RoboDK station: deburring.rdk

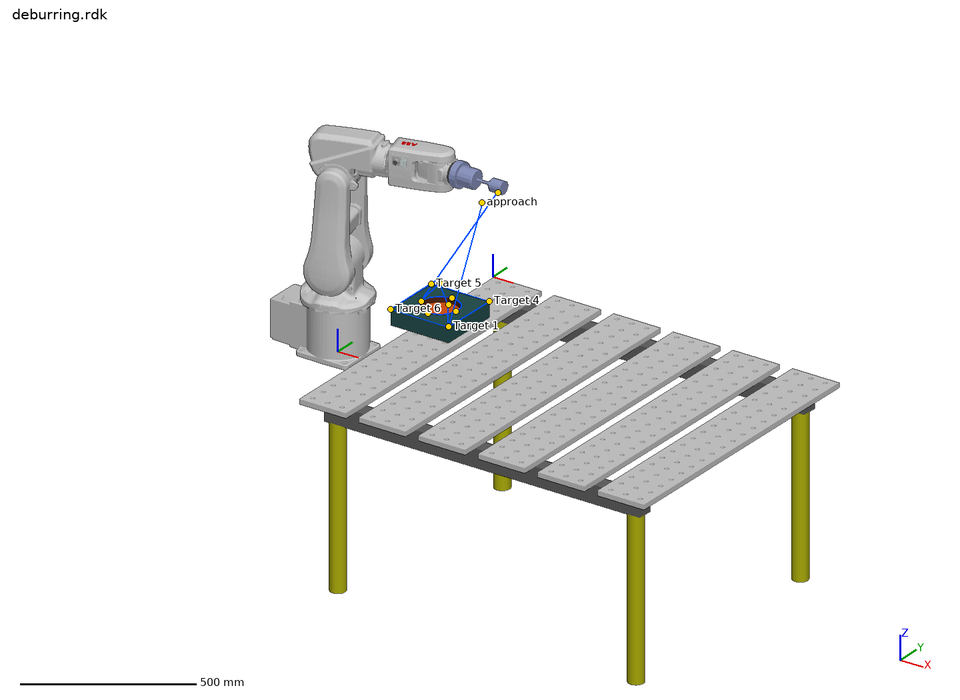
[picture v0: the station drawn from its stored meshes, robots at their saved joint values, targets as dots, program paths as lines]
Station deburring (saved by RoboDK 5.3.4). Poses are relative to the parent item; angles as X-Y-Z fixed-axis rotations.
  - frame ABB IRB 120-3/0.6 Base at (0, 0, 0) mm
    - robot ABB IRB 120-3/0.6: 6 axes, payload 3 kg, reach 580 mm, repeatability 0.01 mm, weight 25 kg
        modified DH rows (alpha deg, a mm, theta deg, d mm): 0, 0, 0, 290; -90, 0, -90, 0; 0, 270, 0, 0; -90, 70, 0, 302; 90, 0, 0, 0; -90, 0, 180, 72
        joint limits [-165, -110, -90, -160, -120, -400] to [165, 110, 70, 160, 120, 400]; home [0, 0, 0, 0, 0, 0]; saved at [14.502, 2.119, -2.154, 90.135, -14.502, -90.14]
      - tool AssemblySpindleSide, TCP at (20, 0, 125) mm, rotated rx 0 ry 45 rz 0 deg, size 80 x 163 x 80 mm
  - object Table at (800, 0, 100) mm, size 1193.8 x 965.2 x 609.6 mm, geometry from welding_table.sld
  - frame worktable at (200, 480, 100) mm
    - object Task2_Part at (60, -590, 100) mm, rotated rx 90 ry 0 rz 0 deg, size 200 x 50 x 200 mm, geometry from Task2_Part.STEP
    - target approach (Cartesian target) at (299, -480, 510) mm, rotated rx -180 ry 45 rz -180 deg; joints [0, 0, 0, 0, 0, 0] of ABB IRB 120-3/0.6
    - target retract (Cartesian target) at (299, -401.89, 510) mm, rotated rx 180 ry 45 rz 180 deg; joints [14.502, 2.119, -2.154, 90.135, -14.502, -90.14] of ABB IRB 120-3/0.6
    - target Target 1 (Cartesian target) at (260, -590, 150) mm, rotated rx 180 ry 0 rz -180 deg; joints [-18.186, 16.881, 24.041, 66.872, 13.885, -79.329] of ABB IRB 120-3/0.6
    - target Target 4 (Cartesian target) at (260, -390, 150) mm, rotated rx -180 ry 0 rz -180 deg; joints [15.045, 15.786, 25.439, -65.976, 11.593, 76.295] of ABB IRB 120-3/0.6
    - target Target 4-5 turning (Cartesian target) at (260, -390, 150) mm, rotated rx 180 ry 0 rz -90 deg; joints [-4.371, 38.309, -6.748, 48.185, 71.084, -116.089] of ABB IRB 120-3/0.6
    - target Target 5 (Cartesian target) at (60, -390, 150) mm, rotated rx -180 ry 0 rz -90 deg; joints [-7.701, -1.111, 44.482, 50.43, 65.373, -127.586] of ABB IRB 120-3/0.6
    - target Target 5-6 turning (Cartesian target) at (60, -390, 150) mm, rotated rx 180 ry 0 rz 0 deg; joints [13.152, 25.112, 12.943, 9.312, 96.103, -169.619] of ABB IRB 120-3/0.6
    - target Target 6 (Cartesian target) at (60, -590, 150) mm, rotated rx 180 ry 0 rz 0 deg; joints [-15.939, 26.08, 11.574, -11.262, 96.105, -192.63] of ABB IRB 120-3/0.6
    - target Target 6-7 turning (Cartesian target) at (60, -590, 150) mm, rotated rx -180 ry 0 rz 90 deg; joints [3.337, -1.525, 44.887, -52.465, 62.898, -234.62] of ABB IRB 120-3/0.6
    - target Target 7 (Cartesian target) at (260, -590, 150) mm, rotated rx -180 ry 0 rz 90 deg; joints [1.887, 38.076, -6.383, -49.021, 69.41, 114.709] of ABB IRB 120-3/0.6
    - target Target 7 protect (Cartesian target) at (260, -590, 220) mm, rotated rx -180 ry 0 rz 90 deg; joints [1.887, 34.449, -14.133, -46.477, 77.076, 105.92] of ABB IRB 120-3/0.6
    - target Target 8 (Cartesian target) at (160, -490, 220) mm, rotated rx -180 ry 0 rz -180 deg; joints [-2.438, -13.888, 41.637, 5.787, 17.359, -7.249] of ABB IRB 120-3/0.6
    - target Target 13 (Cartesian target) at (100.44, -497.23, 150) mm, rotated rx 180 ry 0 rz 180 deg; joints [-5.615, -22.25, 61.415, 33.679, 7.167, -37.448] of ABB IRB 120-3/0.6
    - target Target 17 (Cartesian target) at (219.56, -497.23, 150) mm, rotated rx -180 ry 0 rz 0 deg; joints [-1.812, 60.736, -44.257, -1.458, 118.499, -181.977] of ABB IRB 120-3/0.6
    - target Target 15 (Cartesian target) at (160, -430, 150) mm, rotated rx -180 ry 0 rz 90 deg; joints [25.945, 26.039, 11.631, -40.337, 79.208, 133.566] of ABB IRB 120-3/0.6
    - target Target 16 (Cartesian target) at (160, -550, 150) mm, rotated rx -180 ry 0 rz -90 deg; joints [-28.462, 27.811, 9.093, 38.995, 81.076, -134.635] of ABB IRB 120-3/0.6
  - program prog1 (15 instructions, listed below)
  - program main (1 instructions, listed below)
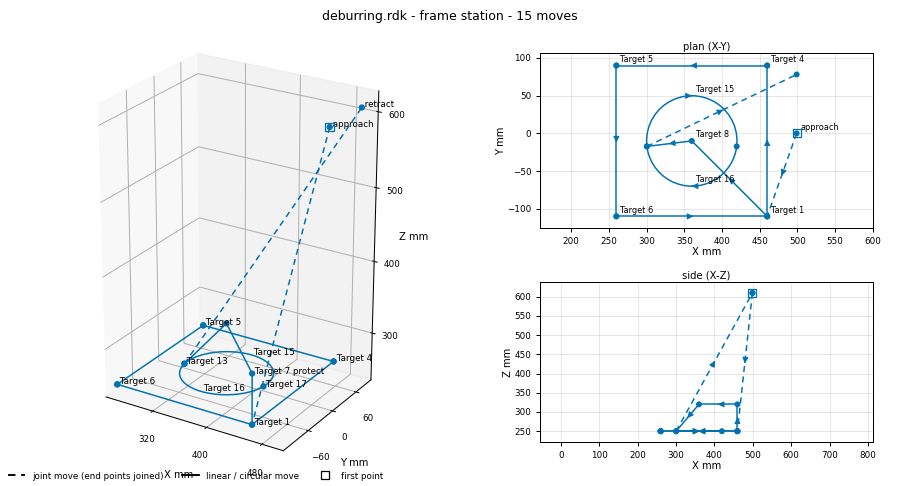
[picture p0: tool path of deburring.rdk in frame station, 15 of 15 moves have a stored position in this frame; points joined in program order, loops and branches not executed]

--- program prog1 (robot ABB IRB 120-3/0.6) ---
  MoveJ (approach)
  MoveJ (Target 1)
  MoveL (Target 4)
  MoveL (Target 4-5 turning)
  MoveL (Target 5)
  MoveL (Target 5-6 turning)
  MoveL (Target 6)
  MoveL (Target 6-7 turning)
  MoveL (Target 7)
  MoveL (Target 7 protect)
  MoveL (Target 8)
  MoveL (Target 13)
  MoveC (Target 15, Target 17)
  MoveC (Target 16, Target 13)
  MoveJ (retract)

--- program main (robot ABB IRB 120-3/0.6) ---
  调用 prog1
